Staubli VAL3: GetPostion.pjx

--- GetPostion.pjx ---
Parameters version=s7.9 stackSize=5000 millimeterUnit=true
Program file=Move.pgx
Program file=Postion.pgx
Program file=View.pgx
Program file=start.pgx
Program file=stop.pgx
Data file=GetPostion.dtx

--- start.pgx ---
program start()
begin
  //2016.07.01
  //三个任务
  //1. 运动
  //2. 获取当前位置
  //3. 人机界面


  // call View()
  //异步任务
  taskCreate "move",100,Move()
  taskCreate "View",100,View()

  taskCreateSync "postion",0.004,bOver,Postion()






end

--- Postion.pgx ---
program Postion()
  local num l_nStart
  local string l_sBuff
  local num l_nNum
begin

  //运动堆栈不为空
  wait(!isEmpty())

  l_nStart=clock()

  //先关掉所有文件
  //保证每次只操作一个文件
  $fileClose(0)
  $fileClose(1)
  $fileClose(2)
  $fileClose(3)
  $fileClose(4)
  $fileClose(5)
  $fileClose(6)
  $fileClose(7)
  $fileClose(8)
  $fileClose(9)




  nFileID=$fileOpen("Disk://postion.txt","w")
  if nFileID<0 or nFileID>9
    popUpMsg("文件错误")
    return
  endIf


  l_nNum=0

  while isEmpty()==false

    //获取当前关节位置
    jNow=herej()

    //获取当前坐标系位置
    pNow=here(tTool,world)
    getJointForce(nJointForce)
    if l_nNum<1000
      nForceData[l_nNum,0]=nJointForce[0]
      nForceData[l_nNum,1]=nJointForce[1]
      nForceData[l_nNum,2]=nJointForce[2]
      nForceData[l_nNum,3]=nJointForce[3]
      nForceData[l_nNum,4]=nJointForce[4]
      nForceData[l_nNum,5]=nJointForce[5]
    endIf


    l_nNum=l_nNum+1
    l_sBuff=toString(".3",jNow.j1)+","+toString(".3",jNow.j2)+","+toString(".3",jNow.j3)+","
    l_sBuff=l_sBuff+toString(".3",jNow.j4)+","+toString(".3",jNow.j5)+","+toString(".3",jNow.j6)+","
    l_sBuff=l_sBuff+toString(".3",pNow.trsf.x)+","+toString(".3",pNow.trsf.y)+","+toString(".3",pNow.trsf.z)+","
    l_sBuff=l_sBuff+toString(".3",pNow.trsf.rx)+","+toString(".3",pNow.trsf.ry)+","+toString(".3",pNow.trsf.rz)+","
    l_sBuff=l_sBuff+toString(".3",clock()-l_nStart)+","+toString("",l_nNum)




    if $fileSet(nFileID,l_sBuff,1)!=1
      popUpMsg("error")
      return
    endIf



    delay(0)
  endWhile

  for l_nNum=0 to 9999


 endFor




  $fileClose(0)
  $fileClose(1)
  $fileClose(2)
  $fileClose(3)
  $fileClose(4)
  $fileClose(5)
  $fileClose(6)
  $fileClose(7)
  $fileClose(8)
  $fileClose(9)


 popUpMsg("运行时间："+toString(".3",clock()-l_nStart))










end

--- View.pgx ---
program View()
begin
  //显示出结果
  //清屏
  cls()
  //跳到用户界面
  userPage()


  gotoxy(0,0)
  put("机械手臂当前位置:")

  while true
    gotoxy(0,1)
    put("J1:"+toString(".3",jNow.j1)+"      ")

    gotoxy(0,2)
    put("J2:"+toString(".3",jNow.j2)+"      ")

    gotoxy(0,3)
    put("J3:"+toString(".3",jNow.j3)+"      ")
    gotoxy(0,4)
    put("J4:"+toString(".3",jNow.j4)+"      ")
    gotoxy(0,5)
    put("J5:"+toString(".3",jNow.j5)+"      ")
    gotoxy(0,6)
    put("J6:"+toString(".3",jNow.j6)+"      ")


    //坐标系

    gotoxy(0,7)
    put("X:"+toString(".3",pNow.trsf.x)+"      ")

    gotoxy(0,8)
    put("Y:"+toString(".3",pNow.trsf.y)+"      ")

    gotoxy(0,9)
    put("Z:"+toString(".3",pNow.trsf.z)+"      ")

    gotoxy(0,10)
    put("RX:"+toString(".3",pNow.trsf.rx)+"      ")

    gotoxy(0,11)
    put("RY:"+toString(".3",pNow.trsf.ry)+"      ")
    gotoxy(0,12)
    put("RZ:"+toString(".3",pNow.trsf.rz)+"      ")




    delay(0)


  endWhile









end
